FUNCTION INTERNAL F_IncrementStep
VAR_IN_OUT
	nStepToInc : INT; 
END_VAR
VAR_IN_OUT CONSTANT
	sActiveStep : T_MaxString; 
END_VAR
VAR_INPUT
	eMode : E_Mode;
END_VAR
VAR CONSTANT
	cStepFinished : INT := -999;
END_VAR

CASE eMode OF
	E_Mode.BUSY:
		RETURN;
	E_Mode.INC:
		nStepToInc := nStepToInc + 1;
		IF sActiveStep <> '' THEN
			TEST_FINISHED_NAMED(sActiveStep);
		END_IF
	E_Mode.END:
		nStepToInc := cStepFinished;
		IF sActiveStep <> '' THEN
			TEST_FINISHED_NAMED(sActiveStep);
		END_IF
END_CASE

END_FUNCTION

(* stored: Version 1.1.0.1, ProductVersion 3.1.4024.12
   POU F_IncrementStep: Id {701464ed-4ab7-4ccb-a3fd-1cc65c5b3c94}, SpecialFunc None *)
